TEXTLIST FiX_1
  0 = 'CYCLE START'
  10 = 'RD_CLOSE'
  20 = 'TRUNION ROTATES -20*'
  30 = 'RD OPEN'
  40 = 'OPERATOR LOAD 1ST PART'
  50 = 'OPERATOR LOAD 2ND PART'
  60 = 'Clamp Close_1ST,3RD,5TH'
  70 = 'RD_CLOSE'
  80 = 'TRUNION ROTATES -80*'
  90 = 'RD OPEN'
  100 = ' Operator Load_3RD_PART'
  110 = ' Operator Load_4TH_PART'
  120 = 'RD_CLOSE'
  130 = ' CLAMP CLOSE 2ND,4TH, 6TH'
  140 = 'TURNTABLE-180* AND TRUNION_0*'
  150 = 'Start WELD_Robot FOR WELD'
  160 = 'CLAMP OPEN 1ST,3RD,5TH'
  170 = 'RD OPEN'
  180 = 'Start MH_Robot_1ST TIME'
  190 = 'TRUNION ROTATES -45*'
  200 = 'UNCLAMP 2ND, 4TH,6TH'
  210 = 'Start MH_Robot_2ND TIME'
  220 = 'CYCLE COMPLETE'
   = ''
END_TEXTLIST

(* stored: Version 1.1.0.1, ProductVersion 3.1.4024.16
   TextList FiX_1: Id {5fb94b9e-8a1a-427b-be9e-ac42e447a106} *)
